// Mitsubishi GX Works2 project: 2023-05-18 #1 생산자동화기능사 1번   PLC: Q03UDV
// 생산자동화기능사

// global labels: Global1
VAR_GLOBAL
  PB1 AT X0 : BOOL;
  PB2 AT X1 : BOOL;
  정지 AT X2 : BOOL;
  공급후진 AT X3 : BOOL;
  공급전진 AT X4 : BOOL;
  가공후진 AT X5 : BOOL;
  가공전진 AT X6 : BOOL;
  송출후진 AT X7 : BOOL;
  송출전진 AT X8 : BOOL;
  배출후진 AT X9 : BOOL;
  배출전진 AT X0A : BOOL;
  매거진 AT X0B : BOOL;
  금속센서 AT X0F : BOOL;
  PB3 AT X0C : BOOL;
  적색 AT Y20 : BOOL;
  황색 AT Y21 : BOOL;
  녹색 AT Y22 : BOOL;
  공급1 AT Y23 : BOOL;
  공급2 AT Y24 : BOOL;
  가공 AT Y25 : BOOL;
  드릴 AT Y26 : BOOL;
  송출 AT Y27 : BOOL;
  배출 AT Y28 : BOOL;
  컨베이어 AT Y29 : BOOL;
END_VAR

PROGRAM 테스트동작
VAR
  STATE : INT;
END_VAR
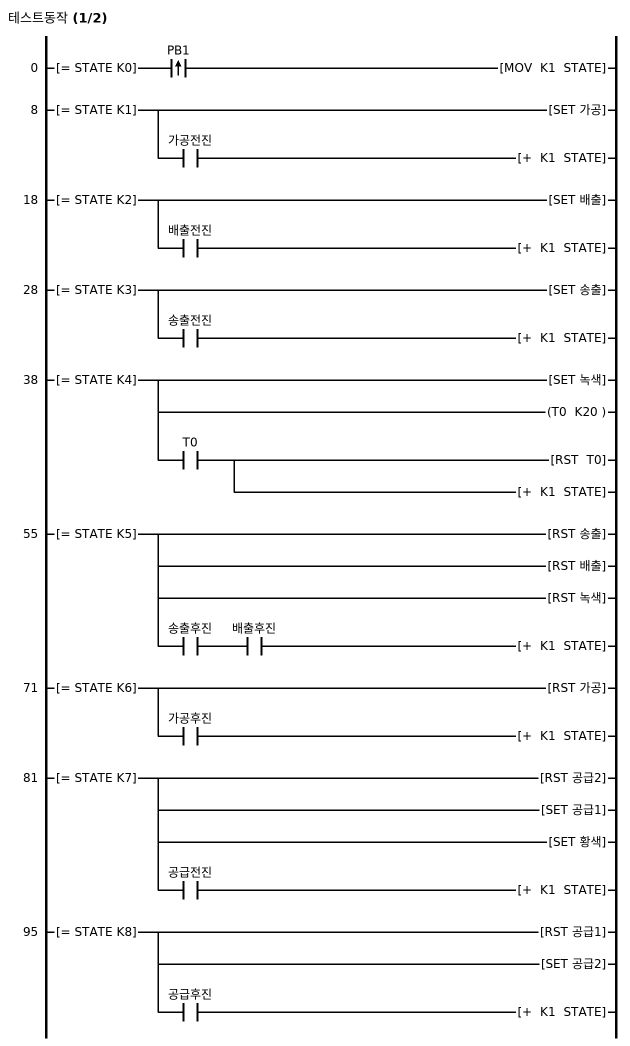
0     LD=     STATE K0
      ANDP    PB1
      MOV     K1 STATE
8     LD=     STATE K1
      SET     가공
      AND     가공전진
      +       K1 STATE
18    LD=     STATE K2
      SET     배출
      AND     배출전진
      +       K1 STATE
28    LD=     STATE K3
      SET     송출
      AND     송출전진
      +       K1 STATE
38    LD=     STATE K4
      SET     녹색
      OUT     T0 K20
      AND     T0
      RST     T0
      +       K1 STATE
55    LD=     STATE K5
      RST     송출
      RST     배출
      RST     녹색
      AND     송출후진
      AND     배출후진
      +       K1 STATE
71    LD=     STATE K6
      RST     가공
      AND     가공후진
      +       K1 STATE
81    LD=     STATE K7
      RST     공급2
      SET     공급1
      SET     황색
      AND     공급전진
      +       K1 STATE
95    LD=     STATE K8
      RST     공급1
      SET     공급2
      AND     공급후진
      +       K1 STATE
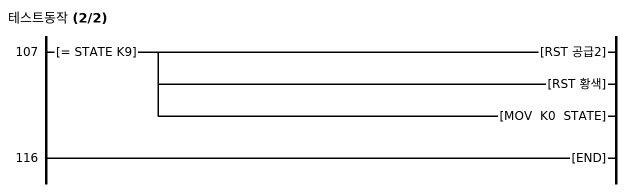
107   LD=     STATE K9
      RST     공급2
      RST     황색
      MOV     K0 STATE
116   END
END_PROGRAM

PROGRAM 단속연속동작
VAR
  STATE : INT;
  MODE : INT;
END_VAR
VAR CONSTANT
  단속 : INT;
  연속 : INT := 1;
END_VAR
VAR
  METAL : BOOL;
  FR1 : ARRAY [0..3] OF BOOL;
  LOOP1 : INT;
  EMSTP : INT;
  FR2 : ARRAY [0..3] OF BOOL;
END_VAR
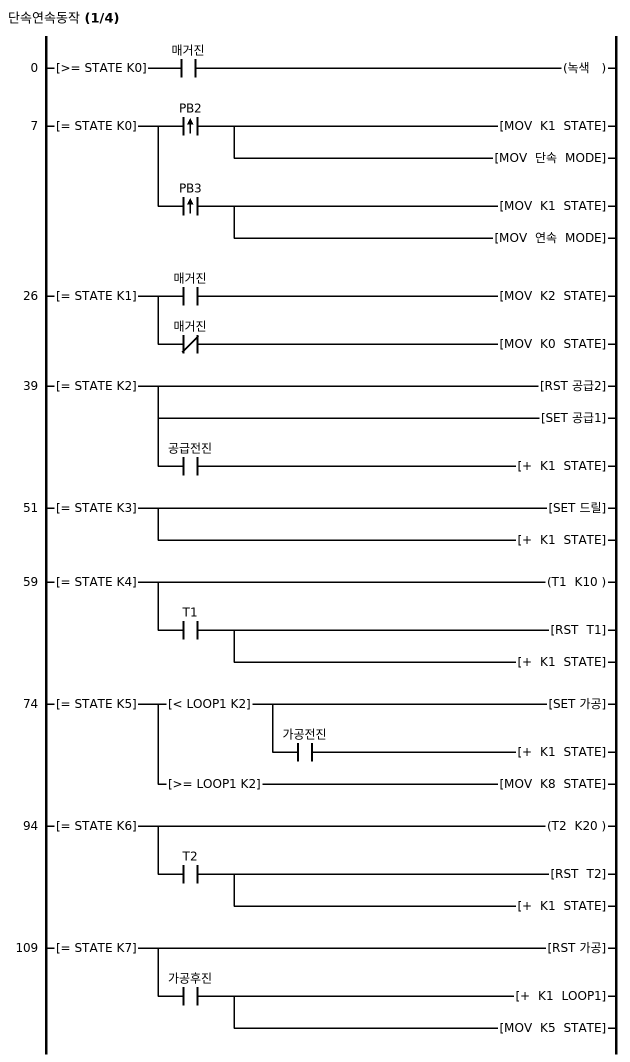
0     LD>=    STATE K0
      AND     매거진
      OUT     녹색
7     LD=     STATE K0
      MPS
      ANDP    PB2
      MOV     K1 STATE
      MOV     단속 MODE
      MPP
      ANDP    PB3
      MOV     K1 STATE
      MOV     연속 MODE
26    LD=     STATE K1
      MPS
      AND     매거진
      MOV     K2 STATE
      MPP
      ANI     매거진
      MOV     K0 STATE
39    LD=     STATE K2
      RST     공급2
      SET     공급1
      AND     공급전진
      +       K1 STATE
51    LD=     STATE K3
      SET     드릴
      +       K1 STATE
59    LD=     STATE K4
      OUT     T1 K10
      AND     T1
      RST     T1
      +       K1 STATE
74    LD=     STATE K5
      MPS
      AND<    LOOP1 K2
      SET     가공
      AND     가공전진
      +       K1 STATE
      MPP
      AND>=   LOOP1 K2
      MOV     K8 STATE
94    LD=     STATE K6
      OUT     T2 K20
      AND     T2
      RST     T2
      +       K1 STATE
109   LD=     STATE K7
      RST     가공
      AND     가공후진
      +       K1 LOOP1
      MOV     K5 STATE
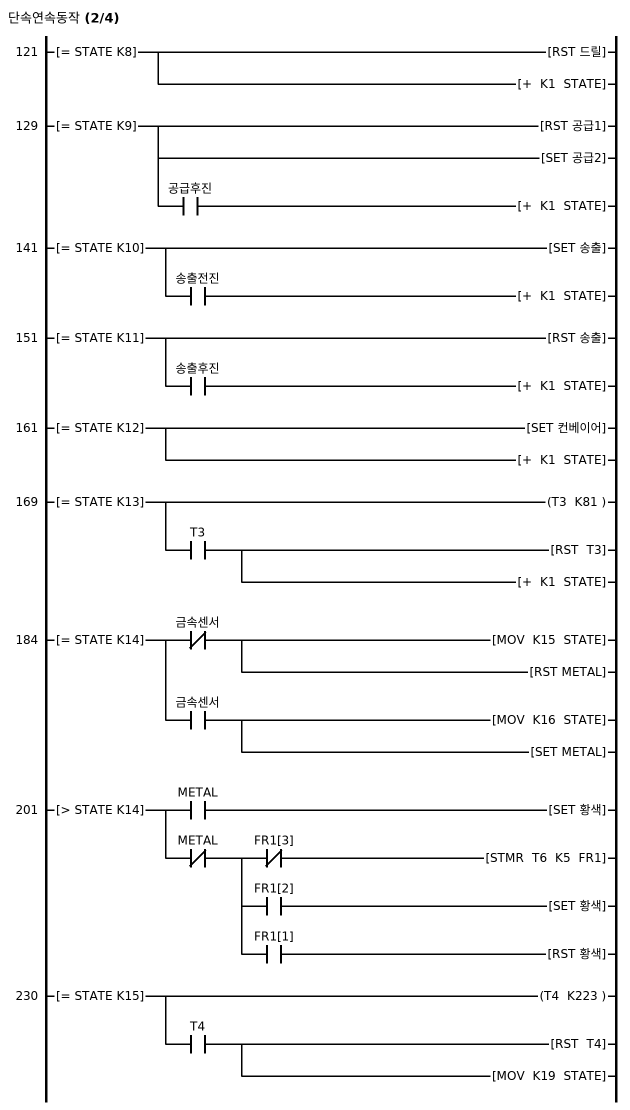
121   LD=     STATE K8
      RST     드릴
      +       K1 STATE
129   LD=     STATE K9
      RST     공급1
      SET     공급2
      AND     공급후진
      +       K1 STATE
141   LD=     STATE K10
      SET     송출
      AND     송출전진
      +       K1 STATE
151   LD=     STATE K11
      RST     송출
      AND     송출후진
      +       K1 STATE
161   LD=     STATE K12
      SET     컨베이어
      +       K1 STATE
169   LD=     STATE K13
      OUT     T3 K81
      AND     T3
      RST     T3
      +       K1 STATE
184   LD=     STATE K14
      MPS
      ANI     금속센서
      MOV     K15 STATE
      RST     METAL
      MPP
      AND     금속센서
      MOV     K16 STATE
      SET     METAL
201   LD>     STATE K14
      MPS
      AND     METAL
      SET     황색
      MPP
      ANI     METAL
      MPS
      ANI     FR1[3]
      STMR    T6 K5 FR1
      MRD
      AND     FR1[2]
      SET     황색
      MPP
      AND     FR1[1]
      RST     황색
230   LD=     STATE K15
      OUT     T4 K223
      AND     T4
      RST     T4
      MOV     K19 STATE
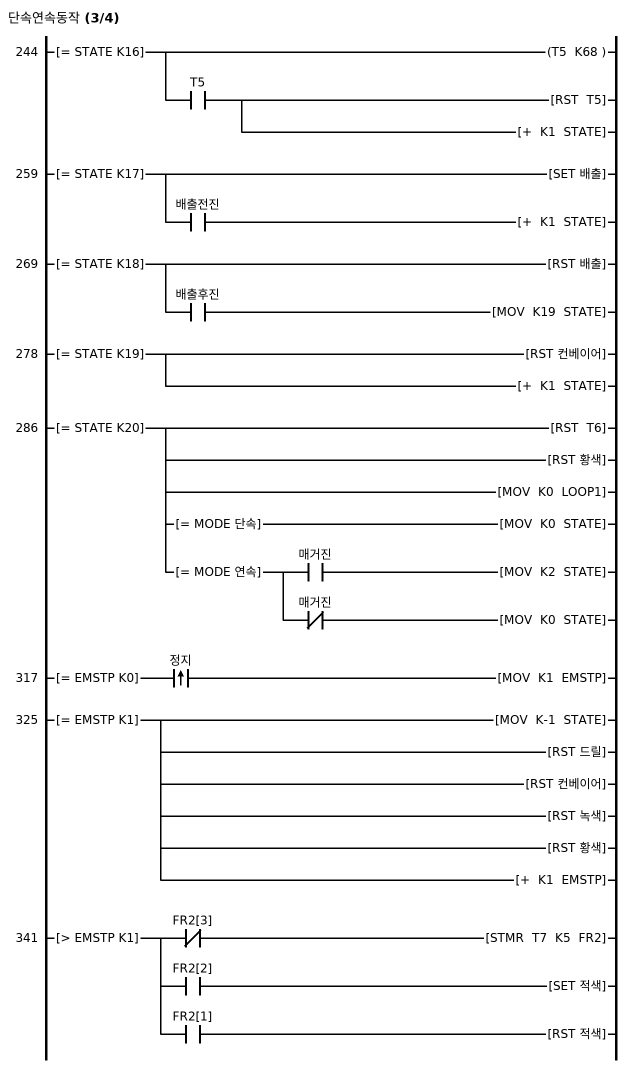
244   LD=     STATE K16
      OUT     T5 K68
      AND     T5
      RST     T5
      +       K1 STATE
259   LD=     STATE K17
      SET     배출
      AND     배출전진
      +       K1 STATE
269   LD=     STATE K18
      RST     배출
      AND     배출후진
      MOV     K19 STATE
278   LD=     STATE K19
      RST     컨베이어
      +       K1 STATE
286   LD=     STATE K20
      RST     T6
      RST     황색
      MOV     K0 LOOP1
      MPS
      AND=    MODE 단속
      MOV     K0 STATE
      MPP
      AND=    MODE 연속
      MPS
      AND     매거진
      MOV     K2 STATE
      MPP
      ANI     매거진
      MOV     K0 STATE
317   LD=     EMSTP K0
      ANDP    정지
      MOV     K1 EMSTP
325   LD=     EMSTP K1
      MOV     K-1 STATE
      RST     드릴
      RST     컨베이어
      RST     녹색
      RST     황색
      +       K1 EMSTP
341   LD>     EMSTP K1
      MPS
      ANI     FR2[3]
      STMR    T7 K5 FR2
      MRD
      AND     FR2[2]
      SET     적색
      MPP
      AND     FR2[1]
      RST     적색
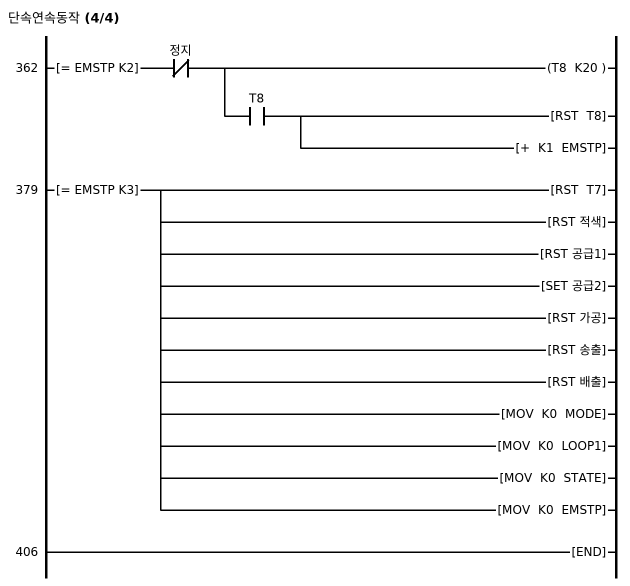
362   LD=     EMSTP K2
      ANI     정지
      OUT     T8 K20
      AND     T8
      RST     T8
      +       K1 EMSTP
379   LD=     EMSTP K3
      RST     T7
      RST     적색
      RST     공급1
      SET     공급2
      RST     가공
      RST     송출
      RST     배출
      MOV     K0 MODE
      MOV     K0 LOOP1
      MOV     K0 STATE
      MOV     K0 EMSTP
406   END
END_PROGRAM
